{attribute 'linkalways'} 
{attribute 'no_explicit_call' := 'This FB is a CLASS and must be accessed using methods or properties'}
{attribute 'enable_dynamic_creation'}
FUNCTION_BLOCK PackML_Mode IMPLEMENTS I_PackML_Mode
VAR
	packMLStateMachine : PackMLStateMachine;
END_VAR

METHOD PUBLIC Abort
VAR_INPUT
END_VAR
packMLStateMachine.Abort();
END_METHOD

METHOD PROTECTED Aborted
VAR_INPUT
	Commands : I_PackML_AbortedCommands;
END_VAR
END_METHOD

METHOD PROTECTED Aborting
VAR_INPUT
	Commands : I_PackML_AbortingCommands;
END_VAR
Commands.StateComplete();
END_METHOD

METHOD PUBLIC Clear
VAR_INPUT
END_VAR
packMLStateMachine.Clear();
END_METHOD

METHOD PROTECTED Clearing
VAR_INPUT
	Commands : I_PackML_ClearningCommands;
END_VAR
Commands.StateComplete();
END_METHOD

METHOD PROTECTED Complete
VAR_INPUT
	Commands : I_PackML_CompleteCommands;
END_VAR
END_METHOD

METHOD PROTECTED Completing
VAR_INPUT
	Commands : I_PackML_CompletingCommands;
END_VAR
Commands.StateComplete();
END_METHOD

PROPERTY PUBLIC CurrentState : PackML_State
GET
CurrentState := packMLStateMachine.CurrentState;
END_GET
END_PROPERTY

METHOD PUBLIC CyclicCall
VAR_INPUT
END_VAR
IF packMLStateMachine.IsIdle THEN 
	Idle(packMLStateMachine);
END_IF

IF packMLStateMachine.IsStarting THEN
	Starting(packMLStateMachine);
END_IF

IF packMLStateMachine.IsExecuting THEN
	Execute(packMLStateMachine);
END_IF

IF packMLStateMachine.IsCompleting THEN
	Completing(packMLStateMachine);
END_IF

IF packMLStateMachine.IsComplete THEN
	Complete(packMLStateMachine);
END_IF

IF packMLStateMachine.IsStopping THEN
	Stopping(packMLStateMachine);
END_IF

IF packMLStateMachine.IsStopped THEN
	Stopped(packMLStateMachine);
END_IF

IF packMLStateMachine.IsResetting THEN
	Resetting(packMLStateMachine);
END_IF

IF packMLStateMachine.IsHolding THEN
	Holding(packMLStateMachine);
END_IF

IF packMLStateMachine.IsHeld THEN
	Held(packMLStateMachine);
END_IF

IF packMLStateMachine.IsUnholding THEN
	Unholding(packMLStateMachine);
END_IF

IF packMLStateMachine.IsSuspending THEN
	Suspending(packMLStateMachine);
END_IF

IF packMLStateMachine.IsSuspended THEN
	Suspended(packMLStateMachine);
END_IF

IF packMLStateMachine.IsUnsuspending THEN
	Unsuspending(packMLStateMachine);
END_IF

IF packMLStateMachine.IsClearing THEN
	Clearing(packMLStateMachine);
END_IF

IF packMLStateMachine.IsAborted THEN
	Aborted(packMLStateMachine);
END_IF

IF packMLStateMachine.IsAborting THEN
	Aborting(packMLStateMachine);
END_IF
END_METHOD

METHOD PROTECTED Execute
VAR_INPUT
	Commands : I_PackML_ExecuteCommands;
END_VAR
Commands.StateComplete();
END_METHOD

METHOD PROTECTED Held
VAR_INPUT
	Commands : I_PackML_HeldCommands;
END_VAR
END_METHOD

METHOD PUBLIC Hold
VAR_INPUT
END_VAR
packMLStateMachine.Hold();
END_METHOD

METHOD PROTECTED Holding
VAR_INPUT
	Commands : I_PackML_HoldingCommands;
END_VAR
Commands.StateComplete();
END_METHOD

METHOD PROTECTED Idle
VAR_INPUT
	Commands : I_PackML_IdleCommands;
END_VAR
END_METHOD

PROPERTY PUBLIC IsAborted : bool
GET
IsAborted := packMLStateMachine.IsAborted;
END_GET
END_PROPERTY

PROPERTY PUBLIC IsAborting : bool
GET
IsAborting := packMLStateMachine.IsAborting;
END_GET
END_PROPERTY

PROPERTY PUBLIC IsClearing : bool
GET
IsClearing := packMLStateMachine.IsClearing;
END_GET
END_PROPERTY

PROPERTY PUBLIC IsComplete : bool
GET
IsComplete := packMLStateMachine.IsComplete;
END_GET
END_PROPERTY

PROPERTY PUBLIC IsCompleting : bool
GET
IsCompleting := packMLStateMachine.IsCompleting;
END_GET
END_PROPERTY

PROPERTY PUBLIC IsExecuting : bool
GET
IsExecuting := packMLStateMachine.IsExecuting;
END_GET
END_PROPERTY

PROPERTY PUBLIC IsHeld : bool
GET
IsHeld := packMLStateMachine.IsHeld;
END_GET
END_PROPERTY

PROPERTY PUBLIC IsHolding : bool
GET
IsHolding := packMLStateMachine.IsHolding;
END_GET
END_PROPERTY

PROPERTY PUBLIC IsIdle : BOOL
GET
isIdle := packMLStateMachine.isIdle;
END_GET
END_PROPERTY

METHOD PUBLIC IsModeTransitionAllowed : BOOL
VAR_INPUT
END_VAR
IsModeTransitionAllowedCheck(packMLStateMachine.CurrentState);
END_METHOD

METHOD PROTECTED IsModeTransitionAllowedCheck : BOOL
VAR_INPUT
	CurrentState : PackML_State;
END_VAR
IsModeTransitionAllowedCheck := true;
END_METHOD

PROPERTY PUBLIC IsResetting : bool
GET
IsResetting := packMLStateMachine.IsResetting;
END_GET
END_PROPERTY

PROPERTY PUBLIC IsStarting : bool
GET
IsStarting := packMLStateMachine.IsStarting;
END_GET
END_PROPERTY

PROPERTY PUBLIC IsStopped : BOOL
GET
isStopped := packMLStateMachine.isStopped;
END_GET
END_PROPERTY

PROPERTY PUBLIC IsStopping : bool
GET
IsStopping := packMLStateMachine.IsStopping;
END_GET
END_PROPERTY

PROPERTY PUBLIC IsSuspended : bool
GET
IsSuspended := packMLStateMachine.IsSuspended;
END_GET
END_PROPERTY

PROPERTY PUBLIC IsSuspending : bool
GET
IsSuspending := packMLStateMachine.IsSuspending;
END_GET
END_PROPERTY

PROPERTY PUBLIC IsUnholding : bool
GET
IsUnholding := packMLStateMachine.IsUnholding;
END_GET
END_PROPERTY

PROPERTY PUBLIC IsUnsuspending : bool
GET
IsUnsuspending := packMLStateMachine.IsUnsuspending;
END_GET
END_PROPERTY

METHOD PUBLIC Reset
VAR_INPUT
END_VAR
packMLStateMachine.Reset();
END_METHOD

METHOD PROTECTED Resetting
VAR_INPUT
	Commands : I_PackML_ResettingCommands;
END_VAR
Commands.StateComplete();
END_METHOD

METHOD PUBLIC Start
VAR_INPUT
END_VAR
packMLStateMachine.Start();
END_METHOD

METHOD PROTECTED Starting
VAR_INPUT
	Commands : I_PackML_StartingCommands;
END_VAR
Commands.StateComplete();
END_METHOD

METHOD PUBLIC Stop
VAR_INPUT
END_VAR
packMLStateMachine.Stop();
END_METHOD

METHOD PROTECTED Stopped
VAR_INPUT
	Commands : I_PackML_StoppedCommands;
END_VAR
END_METHOD

METHOD PROTECTED Stopping
VAR_INPUT
	Commands : I_PackML_StoppingCommands;
END_VAR
Commands.StateComplete();
END_METHOD

METHOD PUBLIC Suspend
VAR_INPUT
END_VAR
packMLStateMachine.Suspend();
END_METHOD

METHOD PROTECTED Suspended
VAR_INPUT
	Commands : I_PackML_SuspendedCommands;
END_VAR
END_METHOD

METHOD PROTECTED Suspending
VAR_INPUT
	Commands : I_PackML_SuspendingCommands;
END_VAR
Commands.StateComplete();
END_METHOD

METHOD PUBLIC Unhold
VAR_INPUT
END_VAR
packMLStateMachine.Unhold();
END_METHOD

METHOD PROTECTED Unholding
VAR_INPUT
	Commands : I_PackML_UnholdingCommands;
END_VAR
Commands.StateComplete();
END_METHOD

METHOD PUBLIC Unsuspend
VAR_INPUT
END_VAR
packMLStateMachine.Unsuspend();
END_METHOD

METHOD PROTECTED Unsuspending
VAR_INPUT
	Commands : I_PackML_UnsuspendingCommands;
END_VAR
Commands.StateComplete();
END_METHOD

END_FUNCTION_BLOCK

(* stored: Version 1.1.0.1, ProductVersion 3.1.4024.12
   POU PackML_Mode: Id {0e04532f-130e-0cc2-0ef6-064aa3e8d498}, SpecialFunc None
   Folder Properties: Id {79d5fa90-7e27-4471-9860-0a94958b6db0}
   Folder Protected: Id {92356802-3353-0857-08ab-5d3ac250c282}
   Folder Public: Id {10ca33f8-22d4-4fff-ba9a-fe572ffb2aa4}
   Method Abort: Id {ee3faf0d-955a-0e0f-2823-dbfcaed60887}
   Method Aborted: Id {a9d09795-ff90-0ada-31dd-d03450f30eae}
   Method Aborting: Id {3465a8a9-1942-0347-040e-7a6b846103d2}
   Method Clear: Id {374b39ac-325b-062b-1ed7-df7f218eeaa6}
   Method Clearing: Id {ece655d6-764d-08f9-39de-5b91ce637dd3}
   Method Complete: Id {d03819d7-063c-0aa0-3ec5-6e7bda8a5a89}
   Method Completing: Id {ed1789d0-cbaa-09ba-3412-bcbd5582875c}
   Property CurrentState: Id {50cab2c6-c5dc-489e-a8fa-d148ac5a9fd8}
   Get Get: Id {483a60ad-41b7-4787-ba4a-1c524323b7b1}
   Method CyclicCall: Id {25b74d63-7bb6-0aea-212a-fa97bd4edbcb}
   Method Execute: Id {15fdf920-b282-0fda-0bd0-60ed33cbd79e}
   Method Held: Id {37533cc7-65a4-062f-11a9-51db2ec15c73}
   Method Hold: Id {0de718c1-967d-0040-0c6c-c4e9eda97436}
   Method Holding: Id {1567001e-6df5-0d24-2b13-277f32781245}
   Method Idle: Id {74b6eebe-4bac-058f-0c93-f4c389fca210}
   Property IsAborted: Id {108b0f52-df45-4ac1-bde9-e8a70721c469}
   Get Get: Id {646b7848-403c-478d-ad41-f210b86bd8aa}
   Property IsAborting: Id {bf7ec69e-ad2a-4fd2-93c2-ffb4034ae93b}
   Get Get: Id {a0d6c53b-d885-4b06-8e84-7c272650460d}
   Property IsClearing: Id {ee0c1866-3c84-4ab3-8ed3-a23607137d75}
   Get Get: Id {3ae7f602-608e-4b9d-9cf3-1816322f2215}
   Property IsComplete: Id {7ae27dc0-3dae-4a07-a372-71c0b1f71d23}
   Get Get: Id {b031b7fb-af8f-4a71-9452-95aad77346e7}
   Property IsCompleting: Id {cb9e2376-4b75-4a07-9935-8d4caf734c7a}
   Get Get: Id {6d78810f-1ec3-4382-8d4e-954e5514a28e}
   Property IsExecuting: Id {24067805-2f79-4643-be9a-5c322a114e98}
   Get Get: Id {f1b49732-f234-4adb-835b-25c2ec9ea59f}
   Property IsHeld: Id {7bea7c71-80f1-4e9b-bd4e-85afce4dd909}
   Get Get: Id {c36b55ba-8658-4658-9a06-0f61ecd6c488}
   Property IsHolding: Id {a06ec06a-33a2-485e-bb71-8e50bd9bd3f0}
   Get Get: Id {54c168c5-230d-423b-88de-4b8b6b81307a}
   Property IsIdle: Id {f558cb81-b86d-4fd1-827f-dc172e8cae4a}
   Get Get: Id {11798741-d714-4420-bec1-e1bfdf299058}
   Method IsModeTransitionAllowed: Id {de5e5643-53bf-4f8d-b8cb-06b45ad0751c}
   Method IsModeTransitionAllowedCheck: Id {eb4c76db-7ee4-4834-89c5-dbc9bf2efd18}
   Property IsResetting: Id {77b02f45-8a87-423c-8be8-e68f6abdb1bd}
   Get Get: Id {b3a25501-6765-4731-8b1c-64f96c164f6c}
   Property IsStarting: Id {975fbac8-cd7d-46a7-add2-11c425c01690}
   Get Get: Id {f6b313e1-8e4a-433e-b9f5-734dfa261c8c}
   Property IsStopped: Id {f107beeb-1f3d-447d-9fc8-f43301e44868}
   Get Get: Id {b3f921a7-3563-4254-85ca-9f47a8770abe}
   Property IsStopping: Id {2cb45f01-f562-4891-add3-c23df79432e5}
   Get Get: Id {1ef89e7f-1763-436a-81c9-7a05faa98292}
   Property IsSuspended: Id {43a4d158-8940-4b66-8c71-0afb75a455e6}
   Get Get: Id {9ce4ccdc-d8d9-43b2-bf06-e7aa6bad982a}
   Property IsSuspending: Id {76f0e6f6-bb70-4714-843c-70c0946a0ca1}
   Get Get: Id {1df51efb-4cb0-4f1b-8959-2318db269d26}
   Property IsUnholding: Id {6822e98c-968d-4ba6-b972-9cc0f5f1df8e}
   Get Get: Id {54bc0434-9efc-41ae-ac44-d69afe21db0f}
   Property IsUnsuspending: Id {aa698aa9-ffb1-4b1c-b51e-f3e933a23564}
   Get Get: Id {62a8f790-775f-4492-9062-77d80b36bb3f}
   Method Reset: Id {1ee5c847-5f73-0a39-3a24-0d7e56c51acd}
   Method Resetting: Id {d102b4c5-0df1-0f6f-3d75-359c9eed8cfb}
   Method Start: Id {4ce820af-166c-0758-033d-44d7f85d5326}
   Method Starting: Id {c0540d4d-914c-031a-0800-0db0955ca094}
   Method Stop: Id {e74449cc-d527-0881-29b5-35132c06dbec}
   Method Stopped: Id {785a423a-f84a-0498-29d4-502601c60e76}
   Method Stopping: Id {0d3cd7ea-2cc6-0723-1740-e4f6cf8e8ad5}
   Method Suspend: Id {49fd49a0-677e-0dfc-1b76-c79b803c1765}
   Method Suspended: Id {5ecd4801-ad57-05cf-3ed0-7c606087443c}
   Method Suspending: Id {024c1967-974a-0dd6-3dcd-572c7c7795e1}
   Method Unhold: Id {3e660fe0-a51e-06e9-0990-610f7ef870e5}
   Method Unholding: Id {4a73c352-cbd7-0ab0-1342-eebf3bd4c02f}
   Method Unsuspend: Id {1fd1510b-7efd-0428-046c-bf1bda2f597f}
   Method Unsuspending: Id {87688408-be2f-00ec-35f1-9cbf9b817928} *)
